ABB RAPID module: Wobj_wt2b.MOD

MODULE Wobj_wt2b
	! Points are read in order of declaration.
  ! Please do not change the order of points!

  LOCAL PERS robtarget pWobj_O_PointX1:=[[111.4713,-633.0164,610.0501],[0.450290441513062,0.515143632888794,0.620464146137238,-0.383262038230896],[-1,0,-1,0],[9E+09,9E+09,9E+09,9E+09,9E+09,9E+09]];
	LOCAL PERS robtarget pWobj_O_PointX2:=[[338.3702,-621.7568,610.277],[0.450279623270035,0.515151798725128,0.620478391647339,-0.383240610361099],[-1,-1,0,0],[9E+09,9E+09,9E+09,9E+09,9E+09,9E+09]];
	LOCAL PERS robtarget pWobj_O_PointY1:=[[112.9341,-764.5509,609.562],[0.45028230547905,0.515146553516388,0.62048876285553,-0.38322776556015],[-1,0,-1,0],[9E+09,9E+09,9E+09,9E+09,9E+09,9E+09]];

ENDMODULE
